		enum_GravaNomes.eAbreConexao: //abre conexao
			IF fbSQLDatabase2.Connect(INT_TO_UDINT(iNumeroDataBase)) THEN
				IF fbSQLDatabase2.bError THEN
					{error <'Não conseguiu abrir a conexao no banco do bloco FB_IniciaOsBlocosDeConfigDoMotor 1'>}
					IF fbSQLDatabase2.ipTcResult.ipSourceInfo.sName = 'ADSERR_DEVICE_LICENSENOTFOUND' THEN
						// se der isso ele nao fica tentando e gerando uma caralhada de erro pq nao tem a lisença
						eEstadoGrava := enum_GravaNomes.eParado;
					ELSE
						eEstadoGrava := enum_GravaNomes.eAbreConexao;
					END_IF
					
				ELSE
					IF fbSQLDatabase2.bConnected THEN
						eEstadoGrava := enum_GravaNomes.eCriaComando;
						xAberto := TRUE;
					ELSE
						eEstadoGrava := enum_GravaNomes.eFechaConexao;
						xAberto := FALSE;
					END_IF
				END_IF
			END_IF
			
		enum_GravaNomes.eCriaComando:
			IF fbSQLDatabase2.CreateCmd(ADR(fbSqlCommand)) THEN
				IF fbSQLDatabase2.bError THEN
					eEstadoGrava := enum_GravaNomes.eCriaComando;
				ELSE
					eEstadoGrava := enum_GravaNomes.eGravaNomes;
				END_IF
			END_IF
			
		enum_GravaNomes.eGravaNomes:
	
			//UPDATE `geral`.`iluminacaoconfig` SET `Tag` = 'IL' WHERE (`Telerruptor` = '1');
			
			Nome := stPM2100[iIndexGrava].config.sNomeFuncao;
			Tag := CONCAT(CONCAT('P', TO_STRING(iIndexGrava)), ' - ');
		
			IF FindAndReplace(
						pSrcString:= ADR(Nome), 
						pDeleteString:= ADR(Tag), 
						pInsertString:= ADR(Vazio), 
						pDstString:= ADR(Funcao), 
						nDstSize:= SIZEOF(Funcao)) = 0  THEN
						
				Funcao := '';	
			END_IF
						
			arrStr[1] := 'UPDATE dbexcelsior.';
			arrStr[2] := sNomeDataBase;
			arrStr[3] := ' SET Funcao = "';
			arrStr[4] := Funcao;
			arrStr[5] :='" WHERE (Medidor = "';
			arrStr[6] := TO_STRING(iIndexGrava);
			arrStr[7] := '");';
			
			sCmd2 := F_ConcatArray(sArray:= arrStr); 
	
			IF fbSQLCommand.Execute(pSQLCmd := ADR(sCmd2), cbSQLCmd := SIZEOF(sCmd2))
			THEN
				IF fbSQLCommand.bError THEN
					IF fbSQLCommand.ipTcResult.nEventId = 61 THEN
					// Esse erro acontece quando o database não tá criado, nesse caso ele tenta criar
						eEstadoGrava := enum_GravaNomes.eEsperando;
						xCriaTabela := TRUE;
					ELSE
						eEstadoGrava := enum_GravaNomes.eAbreConexao;
					END_IF
					sMensagemErro2 := 'Nao conseguiu a tag';
				ELSE
					sMensagemErro2	:= 'Conseguiu a tag';
				END_IF
				eEstadoGrava := enum_GravaNomes.eFechaConexao;
				iIndexGrava := 0;
			END_IF
			
		enum_GravaNomes.eFechaConexao:
			IF fbSQLDatabase2.Disconnect() THEN
		
				xGrava := FALSE;
				xLe := TRUE;
		
				eEstado := enum_LeituradosNomes.eEsperando;
				
				IF fbSQLDatabase2.bError THEN
					eEstadoGrava := enum_GravaNomes.eEsperando;
				ELSE
					eEstadoGrava := enum_GravaNomes.eEsperando;
					xAberto := FALSE;
				END_IF
			END_IF

END_CASE
END_ACTION

ACTION LeNomes:

CASE eEstado OF
		enum_LeituradosNomes.eEsperando: //Esperando
			IF xLe THEN
				eEstado := enum_LeituradosNomes.eAbreConexao;
			END_IF
			
		
		enum_LeituradosNomes.eAbreConexao: //abre conexao
			IF fbSqlDatabase.Connect(int_to_udint(iNumeroDataBase)) THEN
				IF fbSqlDatabase.bError THEN
					{error <'Não conseguiu abrir a conexao no banco do bloco FB_IniciaOsBlocosDeConfigDoMotor 1'>}
					IF fbSqlDatabase.ipTcResult.ipSourceInfo.sName = 'ADSERR_DEVICE_LICENSENOTFOUND' THEN
						// se der isso ele nao fica tentando e gerando uma caralhada de erro pq nao tem a lisença
						eEstado := enum_LeituradosNomes.eParado;
					ELSE
						eEstado := enum_LeituradosNomes.eAbreConexao;
					END_IF
					
				ELSE
					IF fbSqlDatabase.bConnected THEN
						eEstado := enum_LeituradosNomes.eLeOsNomes;
					END_IF
				END_IF
			END_IF
			
			enum_LeituradosNomes.eLeOsNomes: // le o role
				TagAProcurar		:= sTag1;
				stPara.eParaType	:= E_ExpParameterType.STRING_;
				stPara.nParaSize	:= SIZEOF(TagAProcurar);
				stPara.sParaName	:= 'Tag';
		
				diBaixo	:= LOWER_BOUND(stPM2100, 1);
				diCima		:= UPPER_BOUND(stPM2100, 1);
		
				// set command with placeholder
				sCmd := CONCAT(CONCAT('SELECT * FROM dbexcelsior.', sNomeDataBase), ';');
		
				// call functionblock
				IF fbPLCDBCmd.ExecuteDataReturn
					(
						hDBID := INT_TO_UDINT(iNumeroDataBase),
							pExpression := ADR(sCmd),
							cbExpression := SIZEOF(sCmd),
							pData := ADR(TagAProcurar),
							cbData := SIZEOF(TagAProcurar),
							pParameter := ADR(stPara),
							cbParameter := SIZEOF(stPara),
							nStartIndex := DINT_TO_UDINT(diBaixo),
							nRecordCount := DINT_TO_UDINT(diCima),
							pReturnData := ADR(EstruturaBancoLe),
							cbReturnData := SIZEOF(EstruturaBancoLe),
							pRecords := ADR(nRecords))
				THEN
					IF fbPLCDBCmd.bError THEN
						sMensagemErro1 := 'Nao conseguiu a tag';
						{error <'Não conseguiu ler o banco no bloco FB_IniciaOsBlocosDeConfigDoTelerruptor'>}
					ELSE
						sMensagemErro1	:= 'Conseguiu a tag';
						eEstado			:= enum_LeituradosNomes.eFechaConexao;
		
						FOR j := TO_INT(diBaixo) TO TO_INT(diCima) DO
							Anterior[j+1].config.sNomeFuncao := CONCAT(CONCAT(EstruturaBancoLe[j].Tag, ' - '), EstruturaBancoLe[j].Funcao);
							stPM2100[j+1].config.sNomeFuncao := CONCAT(CONCAT(EstruturaBancoLe[j].Tag, ' - '), EstruturaBancoLe[j].Funcao);
						END_FOR
						
					END_IF
				END_IF
			
			enum_LeituradosNomes.eFechaConexao: // FechaConexao conexao
				IF fbSqlDatabase.Disconnect() THEN
		
					xLe := FALSE;
					xInicia := FALSE;
		
					IF fbSqlDatabase.bError THEN
						{error <'Não conseguiu abrir a conexao no banco do bloco FB_IniciaOsBlocosDeConfigDoMotor 3'>}
						eEstado := enum_LeituradosNomes.eFechaConexao;
					ELSE
						eEstado := enum_LeituradosNomes.eMonitoraTrocaDeNomes;
					END_IF
				END_IF	

			enum_LeituradosNomes.eMonitoraTrocaDeNomes:
				FOR j := TO_INT(diBaixo) TO TO_INT(diCima) DO
					IF (stPM2100[j].config.sNomeFuncao <> Anterior[j].config.sNomeFuncao) THEN
						Anterior[j].config.sNomeFuncao := stPM2100[j].config.sNomeFuncao;
						iIndexGrava := j;
						xGrava := TRUE;
					END_IF
				END_FOR						
END_CASE
END_ACTION

END_FUNCTION_BLOCK

// FBs/MedicaoEnergia/FB_NomesMedidoresSEPAM
FUNCTION_BLOCK FB_NomesMedidoresSEPAM
VAR_IN_OUT
	stSEPAM	: ARRAY[*] OF st_SEPAMS20_Schneider;
END_VAR
VAR_INPUT
	xInicia			: BOOL;
	xCriaTabela		: BOOL;
	iNumeroDataBase	: INT		:= 1;
	sNomeDataBase	: STRING	:= 'nomes';
END_VAR
VAR_OUTPUT
	xOcupado	: BOOL;
END_VAR
VAR
	//Cria table
	rtCria			: R_TRIG;
	xCria			: BOOL;
	fbPLCDBCreate	: FB_PLCDBCreateEvt(sNetID := '', tTimeout := T#30S);
	ColumnInfo : ARRAY[0..2] OF ST_ColumnInfo := [(sName := 'Medidor', eType := E_ColumnType.Integer, nLength := 8, sProperty := 'IDENTITY(1,1)'),
												  (sName := 'Tag', eType := E_ColumnType.NVarChar, nLength := 80, sProperty := 'DEFAULT $'SEMTAG$''),
												  (sName := 'Funcao', eType := E_ColumnType.NVarChar, nLength := 80, sProperty := 'DEFAULT $'NADA$'')];
												  

	//Le os nomes
	xFirstScan		: BOOL := TRUE;
	xLe				: BOOL;
	sCmd			: STRING(1000);
	sTag1			: STRING;
	TagAProcurar	: STRING(80);
	sMensagemErro1	: STRING;
	iIndexGrava		: INT := 0;
	iAux			: DINT;
	diCima			: DINT;
	diBaixo			: DINT;
	nRecords		: UDINT;
	Anterior		: ARRAY[0..999] OF st_PM2100_485_Schneider;
	stPara			: ST_ExpParameter;
	EstruturaBancoLe: ARRAY[0..999] OF stConfigNomeMedidorDB;
	eEstado			: enum_LeituradosNomes := enum_LeituradosNomes.eEsperando;
	fbSQLDatabase	: FB_SQLDatabaseEvt(sNetID := '', tTimeout := T#30S);
	fbPLCDBCmd		: FB_PLCDBCmdEvt(sNetID := '', tTimeout := T#30S);
	
	
	//Gera os Telerruptores
	diParteBaixa		: DINT;
	diParteAlta			: DINT;
	i					: INT;
	xGeraMedidores		: BOOL;
	xEscreve			: BOOL;
	xEscreveAux			: BOOL;
	rtEscrita			: R_TRIG;	
	EstruturaBanco		: ARRAY[0..999] OF stConfigNomeMedidorDB;
	fbPLCDBWrite		: FB_PLCDBWriteEvt(sNetID := '', tTimeout := T#30S); //Bloco para gravar no banco de dados
	ColumnNamesGrava	: ARRAY[0..2] OF STRING(50) := ['Medidor',
														'Tag',
														'Funcao'
														];
	//Grava Nomes Novos
	j				: INT;
	xGrava			: BOOL;
	xAberto			: BOOL;
	sCmd2			: STRING(1000);
	sMensagemErro2	: STRING;
	Nome			: STRING;
	Vazio			: STRING := '';
	Tag				: STRING;
	Funcao			: STRING;
	arrStr			: ARRAY[1..10] OF STRING(255);
	eEstadoGrava	: enum_GravaNomes := enum_GravaNomes.eEsperando;
	fbSqlCommand		: FB_SQLCommandEvt(sNetID := '', tTimeout := T#30S);
	fbSQLDatabase2	: FB_SQLDatabaseEvt(sNetID := '', tTimeout := T#30S);
	
END_VAR



IF xFirstScan THEN
	xLe := TRUE;
	xCriaTabela := TRUE;
END_IF

IF xInicia THEN
	xLe := TRUE;
	eEstado := enum_LeituradosNomes.eEsperando;
END_IF




GeraTabela();
//GeraOsMedidores();
LeNomes();
GravaValores();

xFirstScan := FALSE;

ACTION GeraOsMedidores:

diParteBaixa	:= LOWER_BOUND(stSEPAM, 1);
diParteAlta		:= UPPER_BOUND(stSEPAM, 1);

IF xGeraMedidores THEN

	xEscreve := TRUE;
	rtEscrita(CLK := xEscreve, Q =>);

	IF rtEscrita.q THEN
		xEscreveAux						:= TRUE;
		xOcupado						:= TRUE;
		i := DINT_TO_INT(diParteBaixa);
	END_IF

	IF xEscreveAux THEN
		EstruturaBanco[i].Tag := CONCAT('P', INT_TO_STRING(i+1));
		EstruturaBanco[i].Medidor := INT_TO_DINT(i);
		
		IF fbPLCDBWrite.WriteStruct
		(
			hDBID := INT_TO_UDINT(iNumeroDataBase),
				sTableName := sNomeDataBase,
				pRecord := ADR(EstruturaBanco[i]),
				cbRecord := SIZEOF(EstruturaBanco[i]),
				pColumnNames := ADR(ColumnNamesGrava),
				cbColumnNames := SIZEOF(ColumnNamesGrava))
		THEN
			i := i +1;
		ELSE
			IF fbPLCDBWrite.bError THEN
				IF fbPLCDBWrite.ipTcResult.nEventId = 61 THEN
					xCriaTabela := TRUE;
				END_IF
			END_IF
		END_IF
		
		IF i > diParteAlta THEN
			xOcupado	:= FALSE;
			xEscreve 	:= FALSE;
			rtEscrita(CLK := xEscreve, Q =>);
			xEscreveAux	:= FALSE;
			xGeraMedidores := FALSE;
			i := DINT_TO_INT(diParteBaixa);
			
			xLe := TRUE;
			eEstado := enum_LeituradosNomes.eEsperando;
		END_IF

	END_IF
END_IF
END_ACTION

ACTION GeraTabela:

rtCria(CLK := xCriaTabela, Q =>);

IF rtCria.q THEN
	xCria		:= TRUE;
	xOcupado	:= TRUE;
END_IF

IF xCria THEN

	IF fbPLCDBCreate.Table
		(
			hDBID := INT_TO_UDINT(iNumeroDataBase),
				sTableName := sNomeDataBase,
				pTableCfg := ADR(ColumnInfo),
				cbTableCfg := SIZEOF(ColumnInfo))
	THEN
		xCria		:= FALSE;
		xCriaTabela	:= FALSE;
		xOcupado	:= FALSE;
		xGeraMedidores	:= TRUE;
		i			:= 0;
	END_IF

END_IF
END_ACTION

ACTION GravaValores:
CASE eEstadoGrava OF
		enum_GravaNomes.eEsperando: //Esperando
			IF xGrava THEN
				IF xAberto THEN
					eEstadoGrava := enum_GravaNomes.eCriaComando;
				ELSE
					eEstadoGrava := enum_GravaNomes.eAbreConexao;
				END_IF
				
			END_IF
			
		enum_GravaNomes.eAbreConexao: //abre conexao
			IF fbSQLDatabase2.Connect(INT_TO_UDINT(iNumeroDataBase)) THEN
				IF fbSQLDatabase2.bError THEN
					{error <'Não conseguiu abrir a conexao no banco do bloco FB_IniciaOsBlocosDeConfigDoMotor 1'>}
					IF fbSQLDatabase2.ipTcResult.ipSourceInfo.sName = 'ADSERR_DEVICE_LICENSENOTFOUND' THEN
						// se der isso ele nao fica tentando e gerando uma caralhada de erro pq nao tem a lisença
						eEstadoGrava := enum_GravaNomes.eParado;
					ELSE
						eEstadoGrava := enum_GravaNomes.eAbreConexao;
					END_IF
					
				ELSE
					IF fbSQLDatabase2.bConnected THEN
						eEstadoGrava := enum_GravaNomes.eCriaComando;
						xAberto := TRUE;
					ELSE
						eEstadoGrava := enum_GravaNomes.eFechaConexao;
						xAberto := FALSE;
					END_IF
				END_IF
			END_IF
			
		enum_GravaNomes.eCriaComando:
			IF fbSQLDatabase2.CreateCmd(ADR(fbSqlCommand)) THEN
				IF fbSQLDatabase2.bError THEN
					eEstadoGrava := enum_GravaNomes.eCriaComando;
				ELSE
					eEstadoGrava := enum_GravaNomes.eGravaNomes;
				END_IF
			END_IF
			
		enum_GravaNomes.eGravaNomes:
	
			//UPDATE `geral`.`iluminacaoconfig` SET `Tag` = 'IL' WHERE (`Telerruptor` = '1');
			
			Nome := stSEPAM[iIndexGrava].config.sNomeFuncao;
			Tag := CONCAT(CONCAT('P', TO_STRING(iIndexGrava)), ' - ');
		
			IF FindAndReplace(
						pSrcString:= ADR(Nome), 
						pDeleteString:= ADR(Tag), 
						pInsertString:= ADR(Vazio), 
						pDstString:= ADR(Funcao), 
						nDstSize:= SIZEOF(Funcao)) = 0  THEN
						
				Funcao := '';	
			END_IF
						
			arrStr[1] := 'UPDATE dbexcelsior.';
			arrStr[2] := sNomeDataBase;
			arrStr[3] := ' SET Funcao = "';
			arrStr[4] := Funcao;
			arrStr[5] :='" WHERE (Medidor = "';
			arrStr[6] := TO_STRING(iIndexGrava);
			arrStr[7] := '");';
			
			sCmd2 := F_ConcatArray(sArray:= arrStr); 
	
			IF fbSQLCommand.Execute(pSQLCmd := ADR(sCmd2), cbSQLCmd := SIZEOF(sCmd2))
			THEN
				IF fbSQLCommand.bError THEN
					IF fbSQLCommand.ipTcResult.nEventId = 61 THEN
					// Esse erro acontece quando o database não tá criado, nesse caso ele tenta criar
						eEstadoGrava := enum_GravaNomes.eEsperando;
						xCriaTabela := TRUE;
					ELSE
						eEstadoGrava := enum_GravaNomes.eAbreConexao;
					END_IF
					sMensagemErro2 := 'Nao conseguiu a tag';
				ELSE
					sMensagemErro2	:= 'Conseguiu a tag';
				END_IF
				eEstadoGrava := enum_GravaNomes.eFechaConexao;
				iIndexGrava := 0;
			END_IF
			
		enum_GravaNomes.eFechaConexao:
			IF fbSQLDatabase2.Disconnect() THEN
		
				xGrava := FALSE;
				xLe := TRUE;
		
				eEstado := enum_LeituradosNomes.eEsperando;
				
				IF fbSQLDatabase2.bError THEN
					eEstadoGrava := enum_GravaNomes.eEsperando;
				ELSE
					eEstadoGrava := enum_GravaNomes.eEsperando;
					xAberto := FALSE;
				END_IF
			END_IF

END_CASE
END_ACTION

ACTION LeNomes:

CASE eEstado OF
		enum_LeituradosNomes.eEsperando: //Esperando
			IF xLe THEN
				eEstado := enum_LeituradosNomes.eAbreConexao;
			END_IF
			
		
		enum_LeituradosNomes.eAbreConexao: //abre conexao
			IF fbSqlDatabase.Connect(int_to_udint(iNumeroDataBase)) THEN
				IF fbSqlDatabase.bError THEN
					{error <'Não conseguiu abrir a conexao no banco do bloco FB_IniciaOsBlocosDeConfigDoMotor 1'>}
					IF fbSqlDatabase.ipTcResult.ipSourceInfo.sName = 'ADSERR_DEVICE_LICENSENOTFOUND' THEN
						// se der isso ele nao fica tentando e gerando uma caralhada de erro pq nao tem a lisença
						eEstado := enum_LeituradosNomes.eParado;
					ELSE
						eEstado := enum_LeituradosNomes.eAbreConexao;
					END_IF
					
				ELSE
					IF fbSqlDatabase.bConnected THEN
						eEstado := enum_LeituradosNomes.eLeOsNomes;
					END_IF
				END_IF
			END_IF
			
			enum_LeituradosNomes.eLeOsNomes: // le o role
				TagAProcurar		:= sTag1;
				stPara.eParaType	:= E_ExpParameterType.STRING_;
				stPara.nParaSize	:= SIZEOF(TagAProcurar);
				stPara.sParaName	:= 'Tag';
		
				diBaixo	:= LOWER_BOUND(stSEPAM, 1);
				diCima		:= UPPER_BOUND(stSEPAM, 1);
		
				// set command with placeholder
				sCmd := CONCAT(CONCAT('SELECT * FROM dbexcelsior.', sNomeDataBase), ';');
		
				// call functionblock
				IF fbPLCDBCmd.ExecuteDataReturn
					(
						hDBID := INT_TO_UDINT(iNumeroDataBase),
							pExpression := ADR(sCmd),
							cbExpression := SIZEOF(sCmd),
							pData := ADR(TagAProcurar),
							cbData := SIZEOF(TagAProcurar),
							pParameter := ADR(stPara),
							cbParameter := SIZEOF(stPara),
							nStartIndex := DINT_TO_UDINT(diBaixo-1),
							nRecordCount := DINT_TO_UDINT(diCima),
							pReturnData := ADR(EstruturaBancoLe),
							cbReturnData := SIZEOF(EstruturaBancoLe),
							pRecords := ADR(nRecords))
				THEN
					IF fbPLCDBCmd.bError THEN
						sMensagemErro1 := 'Nao conseguiu a tag';
						{error <'Não conseguiu ler o banco no bloco FB_IniciaOsBlocosDeConfigDoTelerruptor'>}
					ELSE
						sMensagemErro1	:= 'Conseguiu a tag';
						eEstado			:= enum_LeituradosNomes.eFechaConexao;
		
						FOR j := TO_INT(diBaixo) TO TO_INT(diCima) DO
							Anterior[j].config.sNomeFuncao := CONCAT(CONCAT(EstruturaBancoLe[j-129].Tag, ' - '), EstruturaBancoLe[j-129].Funcao);
							stSEPAM[j].config.sNomeFuncao := CONCAT(CONCAT(EstruturaBancoLe[j-129].Tag, ' - '), EstruturaBancoLe[j-129].Funcao);
						END_FOR
						
					END_IF
				END_IF
			
			enum_LeituradosNomes.eFechaConexao: // FechaConexao conexao
				IF fbSqlDatabase.Disconnect() THEN
		
					xLe := FALSE;
					xInicia := FALSE;
		
					IF fbSqlDatabase.bError THEN
						{error <'Não conseguiu abrir a conexao no banco do bloco FB_IniciaOsBlocosDeConfigDoMotor 3'>}
						eEstado := enum_LeituradosNomes.eFechaConexao;
					ELSE
						eEstado := enum_LeituradosNomes.eMonitoraTrocaDeNomes;
					END_IF
				END_IF	

			enum_LeituradosNomes.eMonitoraTrocaDeNomes:
				FOR j := TO_INT(diBaixo) TO TO_INT(diCima) DO
					IF (stSEPAM[j].config.sNomeFuncao <> Anterior[j].config.sNomeFuncao) THEN
						Anterior[j].config.sNomeFuncao := stSEPAM[j].config.sNomeFuncao;
						iIndexGrava := j;
						xGrava := TRUE;
					END_IF
				END_FOR						
END_CASE
END_ACTION

END_FUNCTION_BLOCK

// FBs/MedicaoEnergia/FB_SalvaDadosMedidores
FUNCTION_BLOCK FB_SalvaDadosMedidores
VAR_INPUT
	xCriaTabelas		: BOOL;				// tenta criar a tabela
	iNumeroDataBase		: INT	:= 1;		// id do database
	iMedidor			: INT;
	xMedidorOnline		: BOOL;
	rCorrenteA			: REAL;
	rCorrenteB			: REAL;
	rCorrenteC			: REAL;
	rCorrenteMedia		: REAL;
	stHoraAgora			: TIMESTRUCT;
END_VAR
VAR_OUTPUT
	xOcupado 				: BOOL;
	iEndereco				: INT;
END_VAR
VAR
	//Cria table
	rtCria				: R_TRIG;
	xComecaCriarTabelas	: BOOL;
	fbPLCDBCreate1	: FB_PLCDBCreateEvt(sNetID := '', tTimeout := T#30S);
	
	ColumnInfo1 : ARRAY[0..5] OF ST_ColumnInfo := [	(sName := 'rCorrenteA',	eType := E_ColumnType.REAL_,	nLength := 4),
												(sName := 'rCorrenteB',	eType := E_ColumnType.REAL_,	nLength := 4),
												(sName := 'rCorrenteC',	eType := E_ColumnType.REAL_,	nLength := 4),
												(sName := 'rCorrenteMedia',	eType := E_ColumnType.REAL_,	nLength := 4),
												(sName := 'medidor',	eType := E_ColumnType.Integer, 	nLength := 2),
												(sName := 'timestamps', 	eType := E_ColumnType.DateTime, nLength := 4, sProperty := 'DEFAULT CURRENT_TIMESTAMP ON UPDATE CURRENT_TIMESTAMP')];
												
	//Grava valores
	xEscreve			: BOOL;
	rtEscreve			: R_TRIG;
	tonEscrita			: TON;
	arString			: ARRAY[0..6] OF STRING(255);
	fbSqlCommand		: FB_SQLCommandEvt(sNetID := '', tTimeout := T#30S);
	fbSQLDatabase		: FB_SQLDatabaseEvt(sNetID := '', tTimeout := T#30S);
	sCmd				: STRING(1000);
	sMensagemErro1 		: STRING;
	xAberto 			: BOOL;
	rtComecaEscrever 	: R_TRIG;
	iEstado 			: INT := 1;
	i					: INT;
	
END_VAR

//Criado Por Augusto Cazzanelli para o Projeto Excelsior
IF xLicensaValida651641iih THEN
	GeraTabela();
	
	iEndereco := iMedidor;
	
	rtEscreve(CLK:= stHoraAgora.wMinute MOD 5 = 0, Q=> );
	
	IF rtEscreve.Q THEN
		xEscreve := TRUE;
	END_IF
	
	GravaValores();
END_IF

ACTION GeraTabela:

rtCria(CLK := xCriaTabelas, Q =>);

IF rtCria.q THEN
	xComecaCriarTabelas		:= TRUE;
	xOcupado				:= TRUE;
END_IF

IF xComecaCriarTabelas THEN
		//Cria a tabela com os minutos inidividuais de cada um dos 15 min
		IF fbPLCDBCreate1.Table
			(
				hDBID := INT_TO_UDINT(iNumeroDataBase),
					sTableName := 'corrente',
					pTableCfg := ADR(ColumnInfo1),
					cbTableCfg := SIZEOF(ColumnInfo1))
		THEN
			xComecaCriarTabelas		:= FALSE;
			xCriaTabelas	:= FALSE;
			xOcupado := FALSE;
		END_IF
ELSE
	xOcupado := FALSE;
END_IF
END_ACTION

ACTION GravaValores:

CASE iEstado OF
	1: //Esperando
		IF xEscreve AND xMedidorOnline THEN
			IF xAberto THEN
				iEstado := 3;	//Caso para abrir a conexão
			ELSE
				iEstado := 2;	//Caso em que a conexão já foi aberta
			END_IF
		END_IF
		
	2: //abre conexao
		IF fbSqlDatabase.Connect(int_to_udint(iNumeroDataBase)) THEN
			IF fbSqlDatabase.bError THEN
				IF fbSqlDatabase.ipTcResult.nEventId = 1828 THEN
					// se der isso ele nao fica tentando e gerando uma caralhada de erro pq nao tem a lisença
					iEstado := 0;
				ELSE
					iEstado := 2;
				END_IF
			ELSE
				IF fbSqlDatabase.bConnected THEN
					iEstado := 3;
					xAberto := TRUE;
				ELSE
					iEstado := 5;
					xAberto := FALSE;
				END_IF
			END_IF
		END_IF
		
	3:
		IF fbSqlDatabase.CreateCmd(ADR(fbSqlCommand)) THEN
			IF fbSqlDatabase.bError THEN
				iEstado := 3;
			ELSE
				iEstado := 4;
			END_IF
		END_IF
		
		4: // le o role
		//'INSERT INTO dbexcelsior.minutos(rDemanda1min,medidor) VALUES (rDemanda1min, iMedidor);'	
		
		FOR i := 0 TO 3 DO
			arString[i] := '';
		END_FOR
	
		IF xMedidorOnline THEN
			arString[0] := 'INSERT INTO dbexcelsior.corrente(rCorrenteA,rCorrenteB,rCorrenteC,rCorrenteMedia,medidor) VALUES (';
			arString[1] := CONCAT(TO_STRING(rCorrenteA),',');
			arString[2] := CONCAT(TO_STRING(rCorrenteB),',');
			arString[3] := CONCAT(TO_STRING(rCorrenteC),',');
			arString[4] := CONCAT(TO_STRING(rCorrenteMedia),',');
			arString[5] := CONCAT(TO_STRING(iMedidor),');');
		END_IF

	
		sCmd := F_ConcatArray(sArray:= arString);
		
		IF fbSQLCommand.Execute(pSQLCmd := ADR(sCmd), cbSQLCmd := SIZEOF(sCmd)) THEN
			IF fbSQLCommand.bError THEN
				IF fbSQLCommand.ipTcResult.nEventId = 61 THEN
				// Esse erro acontece quando o database não tá criado, nesse caso ele tenta criar
				iEstado := 1;
					xCriaTabelas := TRUE;
				ELSE
					iEstado := 2;
				END_IF
				sMensagemErro1 := 'Nao conseguiu a tag';
			ELSE
				sMensagemErro1	:= 'Conseguiu a tag';
			END_IF
			iEstado := 5;
			xEscreve			:= FALSE;
		END_IF
		
		
	5: // FechaConexao conexao
			IF fbSqlDatabase.Disconnect() THEN
	
				xEscreve			:= FALSE;
	
				IF fbSqlDatabase.bError THEN
					iEstado := 1;
				ELSE
					iEstado := 1;
					xAberto := FALSE;
				END_IF
			END_IF
END_CASE
END_ACTION

END_FUNCTION_BLOCK

// FBs/Partidas/KPI/FB_KPIPartidasSQL
FUNCTION_BLOCK FB_KPIPartidasSQL
VAR_IN_OUT
	Motores : ARRAY[*] OF st_Partida;
END_VAR
VAR_INPUT
	tTempoDeAmostra : TIME;
	xCriaTabela : BOOL;
	iNumeroDataBase : INT := 1;
	sNomeTabela : STRING := 'KPIMotores';
	stHoraAgora : TIMESTRUCT;
	xFazAgora : BOOL;
END_VAR
VAR_OUTPUT
	xGravando : BOOL;
	iRegistro : INT;
END_VAR
VAR
	iEstado : INT := 1;
	rtCria : R_TRIG;
	xCria : BOOL;
	fbPLCDBCreate : FB_PLCDBCreateEvt(sNetID:='', tTimeout:=T#30S);
	
	ColumnInfo : ARRAY[0..7] OF ST_ColumnInfo := [(sName := 'ID', eType := E_ColumnType.BigInt, nLength := 8, sProperty := 'IDENTITY(1,1)'),
												(sName := 'TAG', eType := E_ColumnType.NVarChar, nLength := 80),
												(sName := 'Desligado', eType := E_ColumnType.REAL_, nLength := 8),
												(sName := 'Ligado', eType := E_ColumnType.REAL_, nLength := 8),
												(sName := 'Emergencia', eType := E_ColumnType.REAL_, nLength := 8),
												(sName := 'Falha', eType := E_ColumnType.REAL_, nLength := 8),
												(sName := 'Interlock', eType := E_ColumnType.REAL_, nLength := 8),
												(
				sName := 'Timestamp',
					eType := E_ColumnType.DateTime,
					nLength := 4,
					sProperty :='DEFAULT CURRENT_TIMESTAMP ON UPDATE CURRENT_TIMESTAMP')];
	
	tonEscrita : TON;
	xEscreve : BOOL;
	
	xAtualiza : BOOL;
	ColumnNames : ARRAY[0..6] OF STRING(50) := ['ID',
												'TAG',
												'Desligado',
												'Ligado',
												'Emergencia',
												'Falha',
												'Interlock'];
	iTamanhoHistorico : DINT;
	
	i : INT;
	
	fbPLCDBWrite : FB_PLCDBWriteEvt(sNetID:='', tTimeout:=T#30S); //Bloco para gravar no banco de dados
	sMensagemErroEscrita : STRING;
	
	AuxEscreve : ARRAY[1..500] OF st_KPISQL;
	
	wHoraAnterior : WORD;
	xFirstScan : BOOL := TRUE;
	iMax : INT;
	iMin : INT;
END_VAR



IF xFirstScan THEN
	iMax := DINT_TO_INT(UPPER_BOUND(Motores,1));
	iMin := DINT_TO_INT(LOWER_BOUND(Motores,1));
	
	wHoraAnterior 	:= stHoraAgora.wHour;
END_IF


IF (stHoraAgora.wHour <> wHoraAnterior AND stHoraAgora.wMinute = 2) OR xFazAgora AND NOT xGravando THEN
	
	FOR i := iMin + 1 TO iMax DO
		IF Motores[i].KPI[1].rPorcDesligado > 0.01 THEN
			AuxEscreve[i].Desligado := Motores[i].KPI[1].rPorcDesligado;
		ELSE
			AuxEscreve[i].Desligado := 0;
		END_IF
		
		IF Motores[i].KPI[1].rPorcEmergencia > 0.01 THEN
			AuxEscreve[i].Emergencia := Motores[i].KPI[1].rPorcEmergencia;
		ELSE
			AuxEscreve[i].Emergencia := 0;
		END_IF
		
		IF Motores[i].KPI[1].rPorcFalha > 0.01 THEN
			AuxEscreve[i].Falha := Motores[i].KPI[1].rPorcFalha;
		ELSE
			AuxEscreve[i].Falha := 0;
		END_IF
		
		IF Motores[i].KPI[1].rPorcInterlock > 0.01 THEN
			AuxEscreve[i].Interlock := Motores[i].KPI[1].rPorcInterlock;
		ELSE
			AuxEscreve[i].Interlock := 0;
		END_IF
		
		IF Motores[i].KPI[1].rPorcLigado > 0.01 THEN
			AuxEscreve[i].Ligado := Motores[i].KPI[1].rPorcLigado;
		ELSE
			AuxEscreve[i].Ligado := 0;
		END_IF
		
		IF Motores[iMax].BancoDeDados.Tag <> '' THEN
			AuxEscreve[i].TAG := Motores[i].BancoDeDados.Tag;
		ELSE
			//se nao tiver tag pula fora pra nao ficar rodando onde nao precisa
			EXIT;
		END_IF
	END_FOR

	wHoraAnterior 	:= stHoraAgora.wHour;
	xEscreve		:= TRUE;
	xFazAgora		:= FALSE;
	xGravando 		:= TRUE;
	iRegistro		:= iMin + 1;
END_IF

IF xGravando AND NOT xEscreve THEN
	iRegistro := iRegistro + 1;
	xEscreve := TRUE;
	IF AuxEscreve[iRegistro].TAG = '' THEN
		xGravando := FALSE;
		xEscreve := FALSE;
	END_IF
END_IF

GeraTabela();
GravaHistorico();


xFirstScan := false;

ACTION GeraTabela:

rtCria(CLK := xCriaTabela, Q =>);

IF rtCria.q THEN
	xCria := TRUE;
END_IF

IF xCria THEN

	IF fbPLCDBCreate.Table(
			hDBID := INT_TO_UDINT(iNumeroDataBase),
			sTableName := sNomeTabela,
			pTableCfg := ADR(ColumnInfo),
			cbTableCfg := SIZEOF(ColumnInfo))
	THEN
		xCria := FALSE;
		xCriaTabela := FALSE;
	END_IF

END_IF
END_ACTION

ACTION GravaHistorico:




IF xEscreve THEN
	IF fbPLCDBWrite.WriteStruct(
			hDBID := int_to_Udint(iNumeroDataBase),
			sTableName := sNomeTabela,
			pRecord := ADR(AuxEscreve[iRegistro]),
			cbRecord := SIZEOF(AuxEscreve[iRegistro]),
			pColumnNames := ADR(ColumnNames),
			cbColumnNames := SIZEOF(ColumnNames))
	THEN
		IF fbPLCDBWrite.bError THEN
			sMensagemErroEscrita := 'Erro ao gravar no banco de dados';
			xEscreve             := FALSE;
		ELSE
			sMensagemErroEscrita := 'Dados gravados com sucesso';
			xEscreve             := FALSE;
		END_IF
	END_IF
END_IF
END_ACTION

END_FUNCTION_BLOCK

// FBs/Partidas/SalvaUsoNormal/FB_BDMotores
//{attribute 'hide_all_locals'}
FUNCTION_BLOCK FB_BDMotores
VAR_IN_OUT
	iAtualizandoAtual : INT;
END_VAR
VAR_INPUT
	Motor		: st_Partida;	// st do motor pra pegar os dados
	Nome		: STRING;		// nome do motor para a criação da tabela
	xCriaTabela	: BOOL;			// tenta criar a tabela
	HoraAgora	: TIMESTRUCT;	// pra saber quando gravar
	sCaminhoCSV	: STRING;		// caminho pro CSV
	iMaxAtualizando			: INT := 50;
END_VAR
VAR_OUTPUT
END_VAR
VAR
	// cria tabela
	xCria			: BOOL;
	rtCria			: R_TRIG;
	fbPLCDBCreate	: FB_PLCDBCreateEvt(sNetID := '', tTimeout := T#5S);

	ColumnInfo : ARRAY[0..9] OF ST_ColumnInfo := [(sName := 'ID', eType := E_ColumnType.BigInt, nLength := 8, sProperty := 'IDENTITY(1,1)'),
												(sName := 'Velocidade', eType := E_ColumnType.SmallInt, nLength := 2),
												(sName := 'Corrente', eType := E_ColumnType.REAL_, nLength := 4),
												(sName := 'TemperaturaDoMotor', eType := E_ColumnType.REAL_, nLength := 4),
												(sName := 'Torque', eType := E_ColumnType.REAL_, nLength := 4),
												(sName := 'StatusIHM', eType := E_ColumnType.NVarChar, nLength := 80),
												(sName := 'HorimetroD', eType := E_ColumnType.NVarChar, nLength := 80),
												(sName := 'TotalDePartidas', eType := E_ColumnType.SmallInt, nLength := 2),
												(sName := 'TotalDeFalhas', eType := E_ColumnType.SmallInt, nLength := 2),
												(
				sName := 'Timestamp',
					eType := E_ColumnType.DateTime,
					nLength := 4,
					sProperty := 'DEFAULT CURRENT_TIMESTAMP ON UPDATE CURRENT_TIMESTAMP')];

	// escreve na tabela
	fbPLCDBWrite	: FB_PLCDBWriteEvt(sNetID := '', tTimeout := T#5S);
	ValorPraEscrita	: st_EscritaBD;

	ColumnNames : ARRAY[0..8] OF STRING(50) := ['ID',
												'Velocidade',
												'Corrente',
												'TemperaturaDoMotor',
												'Torque',
												'StatusIHM',
												'HorimetroD',
												'TotalDePartidas',
												'TotalDeFalhas'];

	tUltimoHorimeto	: TIME;
	xEscreve		: BOOL;

	// guarda para escrever o ultimo minuto CSV
	HistoricoDoMinuto : ARRAY[0..59] OF st_EscritaBD;

	rtMudouMinuto	: R_TRIG;
	rtMudouSegundo	: R_TRIG;

	UltimaHora : TIMESTRUCT;

	rtMudouFalhas	: R_TRIG;
	rtMudouPartidas	: R_TRIG;

	iUltimaFalha	: INT;
	iUltimaPartida	: INT;

	rtTrocouDia : R_TRIG;

	//Escrita do CSV
	rtEntrouEmFalha : R_TRIG;

	FBEscreveCSV		: FB_EscreveCSV;
	fbCriaEstruta		: FB_CreateDir;
	dataBase			: ARRAY[0..60, 0..7] OF STRING(255);
	sCaminhoPasta		: STRING;
	sNomeEcaminho		: STRING;
	rtTerminouDeCriar	: R_TRIG;

	sAux : ARRAY[0..25] OF STRING(255);

	i	: INT;
	j	: INT;
	
	xOlhaSeTemEspacoConexao : BOOL;
	rt_TemEspeco : R_TRIG;
	
END_VAR


GeraTabela();

AtualizaValor();

EscreveCSV();

rtMudouMinuto(CLK := tUltimoHorimeto + T#1M = Motor.Sa.tHorimetro, Q =>);

// ve se mudou pra jogar no banco
IF rtMudouMinuto.q AND Motor.Sa.xCmdFwd THEN
	xEscreve		:= TRUE;
	xOlhaSeTemEspacoConexao := FALSE;
	tUltimoHorimeto	:= Motor.Sa.tHorimetro;
END_IF

// se tem espaço pra atualizar ele vai la
rt_TemEspeco(CLK:= xEscreve AND iAtualizandoAtual < iMaxAtualizando, Q=> );
IF rt_TemEspeco.q THEN
	xOlhaSeTemEspacoConexao := TRUE;
	iAtualizandoAtual := iAtualizandoAtual + 1;
END_IF

IF xOlhaSeTemEspacoConexao THEN
	IF fbPLCDBWrite.WriteStruct
		(
			hDBID := 1,
				sTableName := nome,
				pRecord := ADR(ValorPraEscrita),
				cbRecord := SIZEOF(ValorPraEscrita),
				pColumnNames := ADR(ColumnNames),
				cbColumnNames := SIZEOF(ColumnNames))
	THEN
		xEscreve := FALSE;
		xOlhaSeTemEspacoConexao := FALSE;
		iAtualizandoAtual := iAtualizandoAtual - 1;
	END_IF
END_IF

rtMudouSegundo(CLK := HoraAgora.wSecond <> UltimaHora.wSecond, Q =>);

IF rtMudouSegundo.q THEN
	i := WORD_TO_INT(HoraAgora.wSecond);
	HistoricoDoMinuto[i] := ValorPraEscrita;
END_IF

UltimaHora := HoraAgora;

ACTION AtualizaValor:

ValorPraEscrita.Corrente			:= Motor.Sa.rCorrente;
ValorPraEscrita.Velocidade			:= Motor.Sa.iVelocidade;
ValorPraEscrita.TemperaturaDoMotor	:= Motor.Sa.rTemperaturaMotor;
ValorPraEscrita.Torque				:= Motor.Sa.rTorque;

ValorPraEscrita.HorimetroD := Motor.Sa.sHorimetro;

//se tiver em falha ele manda o erro pra BD, se nao manda o status atual dele
IF Motor.Sa.xFalha THEN
	ValorPraEscrita.StatusIHM := Motor.LeiturasInversorIHM.sUltimoErro;
ELSE
	ValorPraEscrita.StatusIHM := Motor.LeiturasInversorIHM.sStatusConexao;
END_IF

// se eles forem diferente e ele for maior que 1 incrementa o numero de falhas, é assim pq o cara pode dar reset no contador
rtMudouFalhas(CLK := ((iUltimaFalha <> Motor.Sa.iFalhaPartida) AND Motor.Sa.iFalhaPartida > 0), Q =>);

IF rtMudouFalhas.q THEN
	ValorPraEscrita.TotalDeFalhas := ValorPraEscrita.TotalDeFalhas + 1;
END_IF

iUltimaFalha := Motor.Sa.iFalhaPartida;

rtMudouPartidas(CLK := (iUltimaPartida <> Motor.Sa.iPartidas) AND Motor.Sa.iPartidas > 0, Q =>);

IF rtMudouPartidas.q THEN
	ValorPraEscrita.TotalDePartidas := ValorPraEscrita.TotalDePartidas + 1;
END_IF

iUltimaPartida := Motor.Sa.iPartidas;

rtTrocouDia(CLK := HoraAgora.wDay <> UltimaHora.wDay, Q =>);

IF rtTrocouDia.q THEN
	ValorPraEscrita.TotalDeFalhas	:= 0;
	ValorPraEscrita.TotalDePartidas	:= 0;
	tUltimoHorimeto					:= Motor.Sa.tHorimetro;
END_IF
END_ACTION

ACTION EscreveCSV:

rtEntrouEmFalha(CLK := Motor.Sa.xFalha AND ValorPraEscrita.StatusIHM <> 'Carregando', Q =>);

IF rtEntrouEmFalha.q THEN
	
	//Pra no segundo de agora pegar a falha
	i := WORD_TO_INT(HoraAgora.wSecond);
	HistoricoDoMinuto[i] := ValorPraEscrita;


	//Ajeita o data base
	dataBase[0, 0]	:= 'Velocidade';
	dataBase[0, 1]	:= 'Corrente';
	dataBase[0, 2]	:= 'TemperaturaDoMotor';
	dataBase[0, 3]	:= 'Torque';
	dataBase[0, 4]	:= 'StatusIHM';
	dataBase[0, 5]	:= 'HorimetroD';
	dataBase[0, 6]	:= 'TotalDePartidas';
	dataBase[0, 7]	:= 'TotalDeFalhas';

	FOR i := 1 TO 60 DO
		FOR J := 0 TO 8 DO
			CASE j OF
				0:
					dataBase[i, j] := TO_STRING(HistoricoDoMinuto[i - 1].Velocidade);

				1:
					dataBase[i, j] := TO_STRING(HistoricoDoMinuto[i - 1].Corrente);

				2:
					dataBase[i, j] := TO_STRING(HistoricoDoMinuto[i - 1].TemperaturaDoMotor);

				3:
					dataBase[i, j] := TO_STRING(HistoricoDoMinuto[i - 1].Torque);

				4:
					dataBase[i, j] := TO_STRING(HistoricoDoMinuto[i - 1].StatusIHM);

				5:
					dataBase[i, j] := TO_STRING(HistoricoDoMinuto[i - 1].HorimetroD);

				6:
					dataBase[i, j] := TO_STRING(HistoricoDoMinuto[i - 1].TotalDePartidas);

				7:
					dataBase[i, j] := TO_STRING(HistoricoDoMinuto[i - 1].TotalDeFalhas);
			END_CASE
		END_FOR
	END_FOR

	//Ve se a pasta ta criada certa 

	fbCriaEstruta(bExecute := TRUE);

	//Ajeita o nome
	sAux[1]			:= sCaminhoCSV;
	sAux[2]			:= '\Falha_';
	sAux[3]			:= Nome;
	sCaminhoPasta	:= CONCAT(sCaminhoCSV, CONCAT('\Falha_', Nome));

	sAux[1]		:= sCaminhoPasta;
	sAux[2]		:= '\';
	sAux[3]		:= TO_STRING(HoraAgora.wYear);
	sAux[4]		:= 'A_';
	sAux[5]		:= TO_STRING(HoraAgora.wMonth);
	sAux[6]		:= 'M_';
	sAux[7]		:= TO_STRING(HoraAgora.wDay);
	sAux[8]		:= 'D_';
	sAux[9]		:= TO_STRING(HoraAgora.wHour);
	sAux[10]	:= 'h_';
	sAux[11]	:= TO_STRING(HoraAgora.wMinute);
	sAux[12]	:= 'm_';
	sAux[13]	:= TO_STRING(HoraAgora.wSecond);
	sAux[20]	:= '.csv';

	sNomeEcaminho := F_ConcatArray(sAux);
END_IF

fbCriaEstruta
	(
		sPathName := sCaminhoPasta,
			ePath := PATH_GENERIC,
			tTimeout := T#5S,
			bBusy =>);

rtTerminouDeCriar(CLK := NOT fbCriaEstruta.bBusy, Q =>);

IF rtTerminouDeCriar.q THEN
	fbCriaEstruta(bExecute := FALSE);
	FBEscreveCSV.bInicia := TRUE;
END_IF

FBEscreveCSV
	(
		sCaminhoENome := sNomeEcaminho,
			xEscrevePorCima := FALSE,
			database := dataBase,
			bBusy =>,
			bError =>,
			nErrId =>,
			iTotal =>,
			iAgora =>);

IF NOT FBEscreveCSV.bBusy THEN
	FBEscreveCSV.bInicia := FALSE;
END_IF
END_ACTION

ACTION GeraTabela:

rtCria(CLK := xCriaTabela, Q =>);

IF rtCria.q THEN
	xCria := TRUE;
END_IF

IF xCria THEN

	IF fbPLCDBCreate.Table
		(
			hDBID := 1,
				sTableName := nome,
				pTableCfg := ADR(ColumnInfo),
				cbTableCfg := SIZEOF(ColumnInfo))
	THEN
		xCria := FALSE;
	END_IF

END_IF
END_ACTION

END_FUNCTION_BLOCK

// FBs/Partidas/FB_CriaTabelaEMotoresParaInterlock
{attribute 'hide_all_locals'}
FUNCTION_BLOCK FB_CriaTabelaEMotoresParaInterlock
VAR_IN_OUT
	Motor : ARRAY[*] OF st_Partida;
END_VAR
VAR_INPUT
	xCriaTabela		: BOOL;
	iNumeroDataBase	: INT		:= 1;
	sNomeDataBase	: STRING	:= 'motoresconfig';
END_VAR
VAR_OUTPUT
	xOcupado : BOOL;
END_VAR
VAR
	i				: INT;
	xGeraMoto		: BOOL;
	diParteBaixa	: DINT;
	diParteAlta		: DINT;

	//Grava valores
	xGravando		: BOOL;
	rtEscrita		: R_TRIG;
	xEscreve		: BOOL;
	EstruturaBanco	: ST_ConfigMotorDB;
	xEscreveAux		: BOOL;
	sAux			: ARRAY[1..50] OF STRING(80);
	fbPLCDBWrite	: FB_PLCDBWriteEvt(sNetID := '', tTimeout := T#30S); //Bloco para gravar no banco de dados

	ColumnNamesGrava : ARRAY[0..27] OF STRING(50) := ['Motor',
														'Tag',
														'Funcao',

														'InvIT1A',
														'IT1A',
														'OPIT1',
														'InvIT1B',
														'IT1B',

														'InvIT2A',
														'IT2A',
														'OPIT2',
														'InvIT2B',
														'IT2B',

														'InvIT3A',
														'IT3A',
														'OPIT3',
														'InvIT3B',
														'IT3B',

														'InvIT4A',
														'IT4A',
														'OPIT4',
														'InvIT4B',
														'IT4B',

														'Emerg1',
														'Emerg2',
														'Emerg3',
														'Emerg4',
														'Timestamp'
														];

	//Cria table
	rtCria			: R_TRIG;
	xCria			: BOOL;
	fbPLCDBCreate	: FB_PLCDBCreateEvt(sNetID := '', tTimeout := T#30S);

	ColumnInfo :
		ARRAY[0..27] OF ST_ColumnInfo
		:= [(sName := 'Motor', eType := E_ColumnType.BigInt, nLength := 8, sProperty := 'IDENTITY(1,1)'),
				(sName := 'Tag', eType := E_ColumnType.NVarChar, nLength := 80, sProperty := 'DEFAULT $'SEMTAG$''),
				(sName := 'Funcao', eType := E_ColumnType.NVarChar, nLength := 80, sProperty := 'DEFAULT $'NADA$''),

				(sName := 'InvIT1A', eType := E_ColumnType.SmallInt, nLength := 2, sProperty := 'DEFAULT 0'),	//Inverte o interlock 1A
				(sName := 'IT1A', eType := E_ColumnType.NVarChar, nLength := 80, sProperty := 'DEFAULT $'-$''),	//TAG do Interlock 1A
				(sName := 'OPIT1', eType := E_ColumnType.SmallInt, nLength := 2, sProperty := 'DEFAULT 0'),		//Operação entre o interlock 1 A e B
				(sName := 'InvIT1B', eType := E_ColumnType.SmallInt, nLength := 2, sProperty := 'DEFAULT 0'),	//Inverte o interlock 1B
				(sName := 'IT1B', eType := E_ColumnType.NVarChar, nLength := 80, sProperty := 'DEFAULT $'-$''),	// TAG do Interlock 1B

				(sName := 'InvIT2A', eType := E_ColumnType.SmallInt, nLength := 2, sProperty := 'DEFAULT 0'),	//Inverte o interlock 2A
				(sName := 'IT2A', eType := E_ColumnType.NVarChar, nLength := 80, sProperty := 'DEFAULT $'-$''),	//TAG do Interlock 2A
				(sName := 'OPIT2', eType := E_ColumnType.SmallInt, nLength := 2, sProperty := 'DEFAULT 0'),		//Operação entre o interlock 2 A e B
				(sName := 'InvIT2B', eType := E_ColumnType.SmallInt, nLength := 2, sProperty := 'DEFAULT 0'),	//Inverte o interlock 2B
				(sName := 'IT2B', eType := E_ColumnType.NVarChar, nLength := 80, sProperty := 'DEFAULT $'-$''),	// TAG do Interlock 2B

				(sName := 'InvIT3A', eType := E_ColumnType.SmallInt, nLength := 2, sProperty := 'DEFAULT 0'),	//Inverte o interlock 3A
				(sName := 'IT3A', eType := E_ColumnType.NVarChar, nLength := 80, sProperty := 'DEFAULT $'-$''),	//TAG do Interlock 3A
				(sName := 'OPIT3', eType := E_ColumnType.SmallInt, nLength := 2, sProperty := 'DEFAULT 0'),		//Operação entre o interlock 3 A e B
				(sName := 'InvIT3B', eType := E_ColumnType.SmallInt, nLength := 2, sProperty := 'DEFAULT 0'),	//Inverte o interlock 3B
				(sName := 'IT3B', eType := E_ColumnType.NVarChar, nLength := 80, sProperty := 'DEFAULT $'-$''),	// TAG do Interlock 3B

				(sName := 'InvIT4A', eType := E_ColumnType.SmallInt, nLength := 2, sProperty := 'DEFAULT 0'),	//Inverte o interlock 4A
				(sName := 'IT4A', eType := E_ColumnType.NVarChar, nLength := 80, sProperty := 'DEFAULT $'-$''),	//TAG do Interlock 4A
				(sName := 'OPIT4', eType := E_ColumnType.SmallInt, nLength := 2, sProperty := 'DEFAULT 0'),		//Operação entre o interlock 4 A e B
				(sName := 'InvIT4B', eType := E_ColumnType.SmallInt, nLength := 2, sProperty := 'DEFAULT 0'),	//Inverte o interlock 4B
				(sName := 'IT4B', eType := E_ColumnType.NVarChar, nLength := 80, sProperty := 'DEFAULT $'-$''),	// TAG do Interlock 4B

				(sName := 'Emerg1', eType := E_ColumnType.NVarChar, nLength := 80, sProperty := 'DEFAULT $'-$''),		//Emergencia 1
				(sName := 'Emerg2', eType := E_ColumnType.NVarChar, nLength := 80, sProperty := 'DEFAULT $'-$''),		//Emergencia 2
				(sName := 'Emerg3', eType := E_ColumnType.NVarChar, nLength := 80, sProperty := 'DEFAULT $'-$''),		//Emergencia 3
				(sName := 'Emerg4', eType := E_ColumnType.NVarChar, nLength := 80, sProperty := 'DEFAULT $'-$''),		//Emergencia 4
			
				
				(
				sName := 'Timestamp',
					eType := E_ColumnType.DateTime,
					nLength := 4,
					sProperty := 'DEFAULT CURRENT_TIMESTAMP ON UPDATE CURRENT_TIMESTAMP')];
END_VAR



IF xLicensaValida651641iih THEN
	
	GeraTabela();
	GeraOsMotores();

END_IF

ACTION GeraOsMotores:

diParteBaixa	:= LOWER_BOUND(Motor, 1);
diParteAlta		:= UPPER_BOUND(Motor, 1);

IF xGeraMoto THEN

	xEscreve := TRUE;
	rtEscrita(CLK := xEscreve, Q =>);

	IF rtEscrita.q THEN
		xEscreveAux						:= TRUE;
		EstruturaBanco.Motor			:= DINT_TO_LINT(diParteBaixa + i);
		EstruturaBanco.Tag				:= CONCAT('MI', TO_STRING(i));
	END_IF

	IF xEscreveAux THEN
		IF fbPLCDBWrite.WriteStruct
			(
				hDBID := INT_TO_UDINT(iNumeroDataBase),
					sTableName := sNomeDataBase,
					pRecord := ADR(EstruturaBanco),
					cbRecord := SIZEOF(EstruturaBanco),
					pColumnNames := ADR(ColumnNamesGrava),
					cbColumnNames := SIZEOF(ColumnNamesGrava))
		THEN
			xEscreve := FALSE;
			rtEscrita(CLK := xEscreve, Q =>);
			xEscreveAux	:= FALSE;
			i			:= i + 1;

			IF i > diParteAlta THEN
				xGeraMoto	:= FALSE;
				xOcupado	:= FALSE;
			END_IF
		ELSE
			IF fbPLCDBWrite.bError THEN
				IF fbPLCDBWrite.ipTcResult.nEventId = 61 THEN
					xCriaTabela := TRUE;
				END_IF
			END_IF
		END_IF
	END_IF

END_IF
END_ACTION

ACTION GeraTabela:

rtCria(CLK := xCriaTabela, Q =>);

IF rtCria.q THEN
	xCria		:= TRUE;
	xOcupado	:= TRUE;
END_IF

IF xCria THEN

	IF fbPLCDBCreate.Table
		(
			hDBID := INT_TO_UDINT(iNumeroDataBase),
				sTableName := sNomeDataBase,
				pTableCfg := ADR(ColumnInfo),
				cbTableCfg := SIZEOF(ColumnInfo))
	THEN
		xCria		:= FALSE;
		xCriaTabela	:= FALSE;
		xGeraMoto	:= TRUE;
		i			:= 1;
	END_IF

END_IF
END_ACTION

END_FUNCTION_BLOCK

// FBs/Sensores/FB_AtualizaTag
{attribute 'hide_all_locals'}
FUNCTION_BLOCK FB_AtualizaTag
VAR_INPUT
	sPayload		: STRING;
	sTag			: STRING;
	iID				: INT;
	xCriaTabela		: BOOL;
	iNumeroDataBase	: INT := 1;
	sNomeDataBase	: STRING;
END_VAR
VAR_OUTPUT
END_VAR
VAR
	//Criar tabela	
	rtCria			: R_TRIG;
	xCria			: BOOL;
	fbPLCDBCreate	: FB_PLCDBCreateEvt(sNetID := '', tTimeout := T#30S);
	ColumnInfo 		: ARRAY[0..3] OF ST_ColumnInfo := [(sName := 'ID', eType := E_ColumnType.BigInt, nLength := 8, sProperty := 'IDENTITY(1,1)'),
													(sName := 'Tag', eType := E_ColumnType.NVarChar, nLength := 80, sProperty := 'DEFAULT $'SEMTAG$''),
													(sName := 'Payload', eType := E_ColumnType.NVarChar, nLength := 80, sProperty := 'DEFAULT $'NADA$''),
													(sName := 'Timestamp', eType := E_ColumnType.DateTime, nLength := 4, sProperty := 'DEFAULT CURRENT_TIMESTAMP ON UPDATE CURRENT_TIMESTAMP')];
												
	//Atualiza									
	xAtualiza : BOOL;	
									
												
	iEstado : INT := 1;
	i : INT;

	sStatusAnterior	: STRING := sPayload;	
	
	arrConcat	: ARRAY[1..15] OF STRING(255);
	arrConcat2	: ARRAY[1..15] OF STRING(255);

	
	fbPLCDBCmd			: FB_PLCDBCmdEvt(sNetID := '', tTimeout := T#30S);
	fbSqlCommand		: FB_SQLCommandEvt(sNetID := '', tTimeout := T#30S);
	fbSQLDatabase		: FB_SQLDatabaseEvt(sNetID := '', tTimeout := T#30S);
	sCmd				: STRING(1000);
	sCmd1				: STRING(255);
	sCmd2				: STRING(255);
	sCmdUpdate			: STRING(1000);
	sMensagemErro1 		: STRING;
	xAberto : BOOL;
	
	FirstScan	: BOOL	:= TRUE;
END_VAR

IF sPayload <> sStatusAnterior THEN
	sStatusAnterior := sPayload;
	xAtualiza := TRUE;
END_IF


IF FirstScan THEN
	xAtualiza := FALSE;
END_IF

GeraTabela();
Atualiza();

FirstScan := FALSE;

ACTION Atualiza:

CASE iEstado OF
	1: //Esperando
		IF xAtualiza THEN
			IF xAberto THEN
				iEstado := 3;
			ELSE
				iEstado := 2;
			END_IF
		END_IF

	2: //abre conexao
		IF fbSqlDatabase.Connect(int_to_udint(iNumeroDataBase)) THEN
			IF fbSqlDatabase.bError THEN
				IF fbSqlDatabase.ipTcResult.nEventId = 1828 THEN
					// se der isso ele nao fica tentando e gerando uma caralhada de erro pq nao tem a lisença
					iEstado := 0;
				ELSE
					iEstado := 2;
				END_IF
			ELSE
				IF fbSqlDatabase.bConnected THEN
					iEstado := 3;
					xAberto := TRUE;
				ELSE
					iEstado := 5;
					xAberto := FALSE;
				END_IF
			END_IF
		END_IF
	
	3:
		IF fbSqlDatabase.CreateCmd(ADR(fbSqlCommand)) THEN
			IF fbSqlDatabase.bError THEN
				iEstado := 3;
			ELSE
				iEstado := 4;
			END_IF
		END_IF
	

	4: // le o role
	
	//UPDATE `maximo`.`sistema` SET `Status` = 'Desligado' WHERE (`ID` = '1');
		
		arrConcat[1] := 'INSERT INTO geral.';
		arrConcat[2] := sNomeDataBase;
		arrConcat[3] := ' (ID,Tag,Payload) VALUES("';
		arrConcat[4] := TO_STRING(iID);
		arrConcat[5] := '","';
		arrConcat[6] := sTag;
		arrConcat[7] := '","';
		arrConcat2[1] := sPayload;
		arrConcat2[2] := '") ON DUPLICATE KEY UPDATE Tag="';
		arrConcat2[3] := sTag;
		arrConcat2[4] := '", Payload="';
		arrConcat2[5] := sPayload;
		arrConcat2[6] := '";';
	
		
		sCmd1 := F_ConcatArray(sArray:= arrConcat);
		sCmd2 := F_ConcatArray(sArray:= arrConcat2);
		
		CONCAT2(pSrcString1:= ADR(sCmd1), pSrcString2:= ADR(sCmd2), pDstString:= ADR(sCmd), nDstSize:= 10000);
		// call functionblock
		IF xAtualiza THEN		
			IF fbSQLCommand.Execute(pSQLCmd := ADR(sCmd), cbSQLCmd := SIZEOF(sCmd))
			THEN
				IF fbSQLCommand.bError THEN
					IF fbSQLCommand.ipTcResult.nEventId = 61 THEN
					// se der isso ele nao fica tentando e gerando uma caralhada de erro pq nao tem a lisença
					iEstado := 1;
						xCriaTabela := TRUE;
					ELSE
						iEstado := 2;
					END_IF
					sMensagemErro1 := 'Nao conseguiu a tag';
				ELSE
					sMensagemErro1	:= 'Conseguiu a tag';
				END_IF
				iEstado := 5;
				xAtualiza := FALSE;
			END_IF
		END_IF

	5: // FechaConexao conexao
		IF fbSqlDatabase.Disconnect() THEN

			xAtualiza := FALSE;

			IF fbSqlDatabase.bError THEN
				iEstado := 1;
			ELSE
				iEstado := 1;
				xAberto := FALSE;
			END_IF
		END_IF
END_CASE
END_ACTION

ACTION GeraTabela:

rtCria(CLK := xCriaTabela, Q =>);

IF rtCria.q THEN
	xCria := TRUE;
END_IF

IF xCria THEN

	IF fbPLCDBCreate.Table(
			hDBID := INT_TO_UDINT(iNumeroDataBase),
			sTableName := sNomeDataBase,
			pTableCfg := ADR(ColumnInfo),
			cbTableCfg := SIZEOF(ColumnInfo))
	THEN
		xCria := FALSE;
		xCriaTabela := FALSE;
	END_IF

END_IF
END_ACTION

END_FUNCTION_BLOCK

// FBs/Sensores/FB_CriaTabelaSensores
{attribute 'hide_all_locals'}
FUNCTION_BLOCK FB_CriaTabelaSensores
VAR_IN_OUT
	Sensores : ARRAY[*] OF st_SensorDigital;
END_VAR
VAR_INPUT
	xCriaTabela		: BOOL;
	iNumeroDataBase	: INT		:= 1;
	sNomeDataBase	: STRING	:= 'SensoresConfig';
	sInicoNome : STRING := 'SO';
END_VAR
VAR_OUTPUT
	xOcupado : BOOL;
END_VAR
VAR
	i				: INT;
	xGeraMoto		: BOOL;
	diParteBaixa	: DINT;
	diParteAlta		: DINT;

	//Grava valores
	xGravando		: BOOL;
	rtEscrita		: R_TRIG;
	xEscreve		: BOOL;
	EstruturaBanco	: st_LeConfigSensorNoBanco;
	xEscreveAux		: BOOL;
	sAux			: ARRAY[1..50] OF STRING(80);
	fbPLCDBWrite	: FB_PLCDBWriteEvt(sNetID := '', tTimeout := T#30S); //Bloco para gravar no banco de dados

	ColumnNamesGrava : ARRAY[0..2] OF STRING(50) := ['Sensor',
													'Tag',
													'Funcao'];

	//Cria table
	rtCria			: R_TRIG;
	xCria			: BOOL;
	fbPLCDBCreate	: FB_PLCDBCreateEvt(sNetID := '', tTimeout := T#30S);

	ColumnInfo :
		ARRAY[0..3] OF ST_ColumnInfo
		:= [(sName := 'Sensor', eType := E_ColumnType.BigInt, nLength := 8, sProperty := 'IDENTITY(1,1)'),
				(sName := 'Tag', eType := E_ColumnType.NVarChar, nLength := 80, sProperty := 'DEFAULT $'SEMTAG$''),
				(sName := 'Funcao', eType := E_ColumnType.NVarChar, nLength := 80, sProperty := 'DEFAULT $'NADA$''),
				(
				sName := 'Timestamp',
					eType := E_ColumnType.DateTime,
					nLength := 4,
					sProperty := 'DEFAULT CURRENT_TIMESTAMP ON UPDATE CURRENT_TIMESTAMP')];
END_VAR

IF xLicensaValida651641iih THEN
	
	GeraTabela();
	GeraOsSensores();
END_IF

ACTION GeraOsSensores:

diParteBaixa	:= LOWER_BOUND(Sensores, 1);
diParteAlta		:= UPPER_BOUND(Sensores, 1);

IF xGeraMoto THEN

	xEscreve := TRUE;
	rtEscrita(CLK := xEscreve, Q =>);

	IF rtEscrita.q THEN
		xEscreveAux						:= TRUE;
		EstruturaBanco.Sensor.dwLowPart	:= DINT_TO_DWORD(diParteBaixa + i);
		EstruturaBanco.Tag				:= CONCAT(sInicoNome, TO_STRING(i));
	END_IF

	IF xEscreveAux THEN
		IF fbPLCDBWrite.WriteStruct
			(
				hDBID := INT_TO_UDINT(iNumeroDataBase),
					sTableName := sNomeDataBase,
					pRecord := ADR(EstruturaBanco),
					cbRecord := SIZEOF(EstruturaBanco),
					pColumnNames := ADR(ColumnNamesGrava),
					cbColumnNames := SIZEOF(ColumnNamesGrava))
		THEN
			xEscreve := FALSE;
			rtEscrita(CLK := xEscreve, Q =>);
			xEscreveAux	:= FALSE;
			i			:= i + 1;

			IF i > diParteAlta THEN
				xGeraMoto	:= FALSE;
				xOcupado	:= FALSE;
			END_IF
		END_IF
	END_IF

END_IF
END_ACTION

ACTION GeraTabela:

rtCria(CLK := xCriaTabela, Q =>);

IF rtCria.q THEN
	xCria		:= TRUE;
	xOcupado	:= TRUE;
END_IF

IF xCria THEN

	IF fbPLCDBCreate.Table
		(
			hDBID := INT_TO_UDINT(iNumeroDataBase),
				sTableName := sNomeDataBase,
				pTableCfg := ADR(ColumnInfo),
				cbTableCfg := SIZEOF(ColumnInfo))
	THEN
		IF NOT fbPLCDBCreate.bError THEN
			xCria		:= FALSE;
			xCriaTabela	:= FALSE;
			xGeraMoto	:= TRUE;
			i			:= 1;
		ELSE
			xCria		:= FALSE;
			xCriaTabela	:= FALSE;
		END_IF
	END_IF

END_IF
END_ACTION

END_FUNCTION_BLOCK

// FBs/Sensores/FB_DBComparaSensor
{attribute 'hide_all_locals'}
FUNCTION_BLOCK FB_DBComparaSensor
VAR_INPUT
	Sensores 		: st_ComparaAnalogico;	// st do sensor analogico lido e manual
	sNomeDataBase	: STRING;				// nome do sensor para a criação da tabela
	iNumeroDataBase	: INT		:= 1;		// id do database	
	xCriaTabela		: BOOL;					// tenta criar a tabela
	tTempoDeAmostra	: TIME;					// tempo entre cada amostra
END_VAR
VAR_OUTPUT
	xOcupado : BOOL;
END_VAR
VAR
	//Cria table
	rtCria			: R_TRIG;
	xCria			: BOOL;
	fbPLCDBCreate	: FB_PLCDBCreateEvt(sNetID := '', tTimeout := T#30S);
	
	ColumnInfo : ARRAY[0..4] OF ST_ColumnInfo := [(sName := 'ID', eType := E_ColumnType.BigInt, nLength := 8, sProperty := 'IDENTITY(1,1)'),
												(sName := 'rAnalogicoLido', eType := E_ColumnType.REAL_, nLength := 4),
												(sName := 'rAnalogicoManual', eType := E_ColumnType.REAL_, nLength := 4),
												(sName := 'rDiferenca', eType := E_ColumnType.REAL_, nLength := 4),
												(
				sName := 'Timestamp',
					eType := E_ColumnType.DateTime,
					nLength := 4,
					sProperty := 'DEFAULT CURRENT_TIMESTAMP ON UPDATE CURRENT_TIMESTAMP')];

	ColumnNamesGrava : ARRAY[0..3] OF STRING(50) := ['ID',
												'rAnalogicoLido',
												'rAnalogicoManual',
												'rDiferenca'];
	
	//Grava valores
	xEscreve			: BOOL;
	fbPLCDBWrite		: FB_PLCDBWriteEvt(sNetID := '', tTimeout := T#30S); //Bloco para gravar no banco de dados
	fbPLCDBCmd			: FB_PLCDBCmdEvt(sNetID := '', tTimeout := T#30S);
	fbSqlCommand		: FB_SQLCommandEvt(sNetID := '', tTimeout := T#30S);
	fbSQLDatabase		: FB_SQLDatabaseEvt(sNetID := '', tTimeout := T#30S);
	sCmd				: STRING(1000);
	sCmdUpdate			: STRING(1000);
	sMensagemErro1 		: STRING;
	xAberto 			: BOOL;
	rtComecaEscrever 	: R_TRIG;
	iEstado 			:	INT := 1;
	tonEscrita			: TON;
	rtSalva				: R_TRIG;
	rAnalogicoManual	: REAL;
	rDiferenca			: REAL;
	xSalva				: BOOL;
END_VAR

IF xLicensaValida651641iih THEN
		
	
	/// Criado por Augusto Cazanelli em 11/05/2022
	
	tonEscrita.IN := TRUE;
	
	rtSalva(CLK:= Sensores.xSalva, Q=> );
	
	IF tonEscrita.q OR rtSalva.Q THEN
		IF (rtSalva.Q) THEN
			rAnalogicoManual := Sensores.rAnalogicoManual;
			xSalva := TRUE;
		ELSE
			rAnalogicoManual := 0;
		END_IF
		
		rDiferenca := Sensores.rAnalogicoLido - rAnalogicoManual; 	
		tonEscrita.IN	:= FALSE;
		xEscreve		:= TRUE;
	END_IF
	
	tonEscrita(PT := tTempoDeAmostra, Q =>, ET =>);
	
	GeraTabela();
	GravaValores();

END_IF

ACTION GeraTabela:

rtCria(CLK := xCriaTabela, Q =>);

IF rtCria.q THEN
	xCria		:= TRUE;
	xOcupado	:= TRUE;
END_IF

IF xCria THEN

	IF fbPLCDBCreate.Table
		(
			hDBID := INT_TO_UDINT(iNumeroDataBase),
				sTableName := sNomeDataBase,
				pTableCfg := ADR(ColumnInfo),
				cbTableCfg := SIZEOF(ColumnInfo))
	THEN
		IF NOT fbPLCDBCreate.bError THEN
			xCria		:= FALSE;
			xCriaTabela	:= FALSE;
		ELSE
			xCria		:= FALSE;
			xCriaTabela	:= FALSE;
		END_IF
	END_IF

END_IF
END_ACTION

ACTION GravaValores:

CASE iEstado OF
	1: //Esperando
		IF xEscreve THEN
			IF xAberto THEN
				iEstado := 3;	//Caso para abrir a conexão
			ELSE
				iEstado := 2;	//Caso em que a conexão já foi aberta
			END_IF
		END_IF

	2: //abre conexao
		IF fbSqlDatabase.Connect(int_to_udint(iNumeroDataBase)) THEN
			IF fbSqlDatabase.bError THEN
				IF fbSqlDatabase.ipTcResult.nEventId = 1828 THEN
					// se der isso ele nao fica tentando e gerando uma caralhada de erro pq nao tem a lisença
					iEstado := 0;
				ELSE
					iEstado := 2;
				END_IF
			ELSE
				IF fbSqlDatabase.bConnected THEN
					iEstado := 3;
					xAberto := TRUE;
				ELSE
					iEstado := 5;
					xAberto := FALSE;
				END_IF
			END_IF
		END_IF
	
	3:
		IF fbSqlDatabase.CreateCmd(ADR(fbSqlCommand)) THEN
			IF fbSqlDatabase.bError THEN
				iEstado := 3;
			ELSE
				iEstado := 4;
			END_IF
		END_IF
	

	4: // le o role
	
		// call functionblock
		IF xEscreve THEN	
		
		IF xSalva THEN
				//'INSERT INTO geral.S01 (rAnalogicoLido, rAnalogicoManual, rDiferenca) VALUES (Sensores.rAnalogicoLido, Sensores.rAnalogicoManual, Sensores.rDiferenca);'	
			sCmd := CONCAT(
					CONCAT(
					CONCAT(
					CONCAT(
					CONCAT(
					CONCAT(
					CONCAT(
					CONCAT(
					'INSERT INTO geral.', sNomeDataBase),
					'(rAnalogicoLido, rAnalogicoManual, rDiferenca) VALUES ('),
					TO_STRING(Sensores.rAnalogicoLido)),
					' , '),
					TO_STRING(rAnalogicoManual)),
					' , '),
					TO_STRING(rDiferenca)),
					');');	
					
					xSalva := FALSE;
		ELSE
							//'INSERT INTO geral.S01 (rAnalogicoLido, rAnalogicoManual, rDiferenca) VALUES (Sensores.rAnalogicoLido, Sensores.rAnalogicoManual, Sensores.rDiferenca);'	
			sCmd := CONCAT(
					CONCAT(
					CONCAT(
					CONCAT(
					CONCAT(
					CONCAT(
					'INSERT INTO geral.', sNomeDataBase),
					'(rAnalogicoLido, rDiferenca) VALUES ('),
					TO_STRING(Sensores.rAnalogicoLido)),
					' , '),
					TO_STRING(rDiferenca)),
					');');	
		END_IF
		
				
			IF fbSQLCommand.Execute(pSQLCmd := ADR(sCmd), cbSQLCmd := SIZEOF(sCmd))
			THEN
				IF fbSQLCommand.bError THEN
					IF fbSQLCommand.ipTcResult.nEventId = 61 THEN
					// Esse erro acontece quando o database não tá criado, nesse caso ele tenta criar
					iEstado := 1;
						xCriaTabela := TRUE;
					ELSE
						iEstado := 2;
					END_IF
					sMensagemErro1 := 'Nao conseguiu a tag';
				ELSE
					sMensagemErro1	:= 'Conseguiu a tag';
				END_IF
				iEstado := 5;
				xEscreve := FALSE;
			END_IF
		END_IF

	5: // FechaConexao conexao
		IF fbSqlDatabase.Disconnect() THEN

			xEscreve := FALSE;

			IF fbSqlDatabase.bError THEN
				iEstado := 1;
			ELSE
				iEstado := 1;
				xAberto := FALSE;
			END_IF
		END_IF
END_CASE
END_ACTION

END_FUNCTION_BLOCK

// FBs/Sensores/FB_HistoricoSQL
{attribute 'hide_all_locals'}
FUNCTION_BLOCK FB_HistoricoSQL
VAR_INPUT
	rValor			: REAL;
	tTempoDeAmostra	: TIME;
	xCriaTabela		: BOOL;
	iNumeroDataBase	: INT := 1;
	sNomeDataBase	: STRING	:= 'LeitorAnalogico1';
END_VAR
VAR_OUTPUT
END_VAR
VAR
	iEstado : INT := 1;
	rtCria			: R_TRIG;
	xCria			: BOOL;
	fbPLCDBCreate	: FB_PLCDBCreateEvt(sNetID := '', tTimeout := T#30S);

	ColumnInfo : ARRAY[0..2] OF ST_ColumnInfo := [(sName := 'ID', eType := E_ColumnType.BigInt, nLength := 8, sProperty := 'IDENTITY(1,1)'),
												(sName := 'Valor', eType := E_ColumnType.Float, nLength := 8),
												(
				sName := 'Timestamp',
					eType := E_ColumnType.DateTime,
					nLength := 4,
					sProperty := 'DEFAULT CURRENT_TIMESTAMP ON UPDATE CURRENT_TIMESTAMP')];


	tonEscrita	: TON;
	xEscreve	: BOOL;


	xAtualiza : BOOL;
	ColumnNamesLe : ARRAY[0..2] OF STRING(50) := ['ID',
												'Valor',
												'Timestamp'];
	iTamanhoHistorico : DINT;

	i : INT;
	
	fbPLCDBCmd			: FB_PLCDBCmdEvt(sNetID := '', tTimeout := T#30S);
	fbSqlCommand		: FB_SQLCommandEvt(sNetID := '', tTimeout := T#30S);
	fbSQLDatabase		: FB_SQLDatabaseEvt(sNetID := '', tTimeout := T#30S);
	sCmd				: STRING(1000);
	sCmdUpdate			: STRING(1000);
	sMensagemErro1 		: STRING;
	xAberto : BOOL;
	rtComecaEscrever : R_TRIG;
END_VAR

IF xLicensaValida651641iih THEN
	

	tonEscrita.IN := TRUE;
	
	IF tonEscrita.q THEN
	tonEscrita.IN	:= FALSE;
	xEscreve		:= TRUE;
	END_IF
	
	tonEscrita(PT := tTempoDeAmostra, Q =>, ET =>);
	
	GeraTabela();
	GravaHistorico();

END_IF

ACTION GeraTabela:

rtCria(CLK := xCriaTabela, Q =>);

IF rtCria.q THEN
	xCria := TRUE;
END_IF

IF xCria THEN

	IF fbPLCDBCreate.Table(
			hDBID := INT_TO_UDINT(iNumeroDataBase),
			sTableName := sNomeDataBase,
			pTableCfg := ADR(ColumnInfo),
			cbTableCfg := SIZEOF(ColumnInfo))
	THEN
		xCria := FALSE;
		xCriaTabela := FALSE;
	END_IF

END_IF
END_ACTION

ACTION GravaHistorico:

CASE iEstado OF
	1: //Esperando
		IF xEscreve THEN
			IF xAberto THEN
				iEstado := 3;
			ELSE
				iEstado := 2;
			END_IF
		END_IF

	2: //abre conexao
		IF fbSqlDatabase.Connect(int_to_udint(iNumeroDataBase)) THEN
			IF fbSqlDatabase.bError THEN
				IF fbSqlDatabase.ipTcResult.nEventId = 1828 THEN
					// se der isso ele nao fica tentando e gerando uma caralhada de erro pq nao tem a lisença
					iEstado := 0;
				ELSE
					iEstado := 2;
				END_IF
			ELSE
				IF fbSqlDatabase.bConnected THEN
					iEstado := 3;
					xAberto := TRUE;
				ELSE
					iEstado := 5;
					xAberto := FALSE;
				END_IF
			END_IF
		END_IF
	
	3:
		IF fbSqlDatabase.CreateCmd(ADR(fbSqlCommand)) THEN
			IF fbSqlDatabase.bError THEN
				iEstado := 3;
			ELSE
				iEstado := 4;
			END_IF
		END_IF
	

	4: // le o role

		sCmd := CONCAT(CONCAT(CONCAT(CONCAT('INSERT INTO geral.', sNomeDataBase),'(Valor) Value ('),TO_STRING(rValor)), ');');	


		// call functionblock
		IF xEscreve THEN		
			IF fbSQLCommand.Execute(pSQLCmd := ADR(sCmd), cbSQLCmd := SIZEOF(sCmd))
			THEN
				IF fbSQLCommand.bError THEN
					IF fbSQLCommand.ipTcResult.nEventId = 61 THEN
					// se der isso ele nao fica tentando e gerando uma caralhada de erro pq nao tem a lisença
					iEstado := 1;
						xCriaTabela := TRUE;
					ELSE
						iEstado := 2;
					END_IF
					sMensagemErro1 := 'Nao conseguiu a tag';
				ELSE
					sMensagemErro1	:= 'Conseguiu a tag';
				END_IF
				iEstado := 5;
				xEscreve := FALSE;
			END_IF
		END_IF

	5: // FechaConexao conexao
		IF fbSqlDatabase.Disconnect() THEN

			xEscreve := FALSE;

			IF fbSqlDatabase.bError THEN
				iEstado := 1;
			ELSE
				iEstado := 1;
				xAberto := FALSE;
			END_IF
		END_IF
END_CASE
END_ACTION

END_FUNCTION_BLOCK

// FBs/Sensores/FB_HistoricoTag
{attribute 'hide_all_locals'}
FUNCTION_BLOCK FB_HistoricoTag
VAR_INPUT
	rValor			: REAL;
	sTag			: STRING;
	tTempoDeAmostra	: TIME;
	xCriaTabela		: BOOL;
	iNumeroDataBase	: INT := 1;
	sNomeDataBase	: STRING;
END_VAR
VAR_OUTPUT
END_VAR
VAR
	//Criar tabela	
	rtCria			: R_TRIG;
	xCria			: BOOL;
	fbPLCDBCreate	: FB_PLCDBCreateEvt(sNetID := '', tTimeout := T#30S);
	ColumnInfo 		: ARRAY[0..2] OF ST_ColumnInfo := [(sName := 'Tag', eType := E_ColumnType.NVarChar, nLength := 80, sProperty := 'DEFAULT $'SEMTAG$''),
													(sName := 'Payload', eType := E_ColumnType.REAL_, nLength := 4),
													(sName := 'Timestamp', eType := E_ColumnType.DateTime, nLength := 4, sProperty := 'DEFAULT CURRENT_TIMESTAMP ON UPDATE CURRENT_TIMESTAMP')];
												
	//Atualiza									
	xAtualiza : BOOL;																		
	iEstado : INT := 1;
	i : INT;
	arrConcat	: ARRAY[1..15] OF STRING(255);
	arrConcat2	: ARRAY[1..15] OF STRING(255);	
	fbPLCDBCmd			: FB_PLCDBCmdEvt(sNetID := '', tTimeout := T#30S);
	fbSqlCommand		: FB_SQLCommandEvt(sNetID := '', tTimeout := T#30S);
	fbSQLDatabase		: FB_SQLDatabaseEvt(sNetID := '', tTimeout := T#30S);
	sCmd				: STRING(1000);
	sCmd1				: STRING(255);
	sCmd2				: STRING(255);
	sCmdUpdate			: STRING(1000);
	sMensagemErro1 		: STRING;
	xAberto 			: BOOL;
	tonEscrita			: Tc2_Standard.TON;
	FirstScan	: BOOL	:= TRUE;
END_VAR


//xAtualiza := TRUE;
tonEscrita.IN := TRUE;

IF tonEscrita.q THEN
	tonEscrita.IN	:= FALSE;
	xAtualiza		:= TRUE;
END_IF

tonEscrita(PT := tTempoDeAmostra, Q =>, ET =>);


IF FirstScan THEN
	xAtualiza := FALSE;
END_IF

GeraTabela();
Atualiza();

FirstScan := FALSE;

ACTION Atualiza:

CASE iEstado OF
	1: //Esperando
		IF xAtualiza THEN
			IF xAberto THEN
				iEstado := 3;
			ELSE
				iEstado := 2;
			END_IF
		END_IF

	2: //abre conexao
		IF fbSqlDatabase.Connect(int_to_udint(iNumeroDataBase)) THEN
			IF fbSqlDatabase.bError THEN
				IF fbSqlDatabase.ipTcResult.nEventId = 1828 THEN
					// se der isso ele nao fica tentando e gerando uma caralhada de erro pq nao tem a lisença
					iEstado := 0;
				ELSE
					iEstado := 2;
				END_IF
			ELSE
				IF fbSqlDatabase.bConnected THEN
					iEstado := 3;
					xAberto := TRUE;
				ELSE
					iEstado := 5;
					xAberto := FALSE;
				END_IF
			END_IF
		END_IF
	
	3:
		IF fbSqlDatabase.CreateCmd(ADR(fbSqlCommand)) THEN
			IF fbSqlDatabase.bError THEN
				iEstado := 3;
			ELSE
				iEstado := 4;
			END_IF
		END_IF
	

	4: // le o role
	
	//UPDATE `maximo`.`sistema` SET `Status` = 'Desligado' WHERE (`ID` = '1');
		
		arrConcat[1] := 'INSERT INTO geral.';
		arrConcat[2] := sNomeDataBase;
		arrConcat[3] := ' (Tag,Payload) VALUES("';
		arrConcat[4] := sTag;
		arrConcat[5] := '",';
		arrConcat2[1] := TO_STRING(rValor);
		arrConcat2[2] := ');';

	
		
		sCmd1 := F_ConcatArray(sArray:= arrConcat);
		sCmd2 := F_ConcatArray(sArray:= arrConcat2);
		
		CONCAT2(pSrcString1:= ADR(sCmd1), pSrcString2:= ADR(sCmd2), pDstString:= ADR(sCmd), nDstSize:= 10000);
		// call functionblock
		IF xAtualiza THEN		
			IF fbSQLCommand.Execute(pSQLCmd := ADR(sCmd), cbSQLCmd := SIZEOF(sCmd))
			THEN
				IF fbSQLCommand.bError THEN
					IF fbSQLCommand.ipTcResult.nEventId = 61 THEN
					// se der isso ele nao fica tentando e gerando uma caralhada de erro pq nao tem a lisença
					iEstado := 1;
						xCriaTabela := TRUE;
					ELSE
						iEstado := 2;
					END_IF
					sMensagemErro1 := 'Nao conseguiu a tag';
				ELSE
					sMensagemErro1	:= 'Conseguiu a tag';
				END_IF
				iEstado := 5;
				xAtualiza := FALSE;
			END_IF
		END_IF

	5: // FechaConexao conexao
		IF fbSqlDatabase.Disconnect() THEN

			xAtualiza := FALSE;

			IF fbSqlDatabase.bError THEN
				iEstado := 1;
			ELSE
				iEstado := 1;
				xAberto := FALSE;
			END_IF
		END_IF
END_CASE
END_ACTION

ACTION GeraTabela:

rtCria(CLK := xCriaTabela, Q =>);

IF rtCria.q THEN
	xCria := TRUE;
END_IF

IF xCria THEN

	IF fbPLCDBCreate.Table(
			hDBID := INT_TO_UDINT(iNumeroDataBase),
			sTableName := sNomeDataBase,
			pTableCfg := ADR(ColumnInfo),
			cbTableCfg := SIZEOF(ColumnInfo))
	THEN
		xCria := FALSE;
		xCriaTabela := FALSE;
	END_IF

END_IF
END_ACTION

END_FUNCTION_BLOCK

// FBs/Sensores/FB_IniciaOsBlocosDeSensor
{attribute 'hide_all_locals'}
FUNCTION_BLOCK FB_IniciaOsBlocosDeSensor
VAR_IN_OUT
	sSensor : ARRAY[*] OF st_SensorDigital;
END_VAR
VAR_INPUT
	xInicia : BOOL;
	iNumeroDataBase	: INT		:= 1;
	sNomeDataBase	: STRING	:= 'SensoresConfig';
END_VAR
VAR_OUTPUT
END_VAR
VAR
	fbPLCDBCmd			: FB_PLCDBCmdEvt(sNetID := '', tTimeout := T#60S);
	fbSQLDatabase		: FB_SQLDatabaseEvt(sNetID := '', tTimeout := T#60S);
	sCmd				: STRING(1000);
	sCmdUpdate			: STRING(1000);
	stPara				: ST_ExpParameter;
	TagAProcurar		: STRING(80);
	nRecords			: UDINT;
	xProcuraNaTabela	: BOOL;
	EstruturaBanco		: ARRAY[0..999] OF Teknike_Sensores.st_LeConfigSensorNoBanco;
	xJogaNoInterlock	: BOOL;
	sTag1				: STRING;
	sTag2				: STRING;
	xEMotor				: BOOL;
	sMensagemErro1		: STRING;
	diCimaSensor		: DINT;
	diBaixoSensor		: DINT;

	iEstado	: INT := 1;
	i		: INT;

	iAux : INT;

END_VAR


IF xLicensaValida651641iih THEN
	
	CASE iEstado OF
		1: //Esperando
			IF xInicia THEN
				iEstado := 2;
			END_IF
	
		2: //abre conexao
			IF fbSqlDatabase.Connect(int_to_udint(iNumeroDataBase)) THEN
				IF fbSqlDatabase.bError THEN
					IF fbSqlDatabase.ipTcResult.ipSourceInfo.sName = 'ADSERR_DEVICE_LICENSENOTFOUND' THEN
						// se der isso ele nao fica tentando e gerando uma caralhada de erro pq nao tem a lisença
						iEstado := 0;
					ELSE
						iEstado := 2;
					END_IF
				ELSE
					IF fbSqlDatabase.bConnected THEN
						iEstado := 3;
					END_IF
				END_IF
			END_IF
	
		3: // le o role
			TagAProcurar		:= sTag1;
			stPara.eParaType	:= E_ExpParameterType.STRING_;
			stPara.nParaSize	:= SIZEOF(TagAProcurar);
			stPara.sParaName	:= 'Tag';
	
			diBaixoSensor	:= LOWER_BOUND(sSensor, 1);
			diCimaSensor	:= UPPER_BOUND(sSensor, 1);
	
			// set command with placeholder
			sCmd := CONCAT(CONCAT('SELECT * FROM ',sNomeDataBase),';');
	
			// call functionblock
			IF fbPLCDBCmd.ExecuteDataReturn
				(
					hDBID := 1,
						pExpression := ADR(sCmd),
						cbExpression := SIZEOF(sCmd),
						pData := ADR(TagAProcurar),
						cbData := SIZEOF(TagAProcurar),
						pParameter := ADR(stPara),
						cbParameter := SIZEOF(stPara),
						nStartIndex := 0,
						nRecordCount := DINT_TO_UDINT(diCimaSensor),
						pReturnData := ADR(EstruturaBanco),
						cbReturnData := SIZEOF(EstruturaBanco),
						pRecords := ADR(nRecords))
			THEN
				IF fbPLCDBCmd.bError THEN
					sMensagemErro1 := 'Nao conseguiu a tag';
				ELSE
					sMensagemErro1	:= 'Conseguiu a tag';
					iEstado			:= 4;
	
					FOR i := TO_INT(diBaixoSensor) TO TO_INT(diCimaSensor)-1 DO
						sSensor[i+1].Banco := EstruturaBanco[i];
						sSensor[i].config.sNome_Funcao := CONCAT(CONCAT(sSensor[i].Banco.Tag,' - '),sSensor[i].Banco.Funcao);
					END_FOR
				END_IF
			END_IF
	
		4: // FechaConexao conexao
			IF fbSqlDatabase.Disconnect() THEN
	
				xInicia := FALSE;
	
				IF fbSqlDatabase.bError THEN
					iEstado := 1;
				ELSE
					iEstado := 1;
				END_IF
			END_IF
	END_CASE

END_IF

END_FUNCTION_BLOCK

// POUs/MAIN
PROGRAM MAIN
VAR
	fb1 : FB_ConfigPartidaNoBanco;
	fb2 : FB_CriaTabelaEMotoresParaInterlock;
	fb3 : FB_IniciaOsBlocosDeConfigDoMotor;
	fb4 : FB_CriaTabelaSensores;
	fb5 : FB_IniciaOsBlocosDeSensor;
	fb6 : FB_HistoricoSQL;
	fb7 : FB_KPIPartidasSQL;
	fb8	: FB_DBComparaSensor;
	fb9	: FB_HistogramaSKUsMaisLidas;
	fb10	: FB_CriaTabelaEmergencias;
	fb11	: FB_IniciaOsBlocosDaEmergencia;
	fb12	: FB_IniciaGrupos;
	fb13	: FB_ControleGrupo;
	fb14	: FB_GeraListaInterlocksIHM;
END_VAR

END_PROGRAM

// Project Information/F_GetCompany
// This function has been automatically generated from the project information.
{attribute 'signature_flag' := '1073741824'}
{attribute 'TcGenerated'}
{attribute 'no-analysis'}
FUNCTION F_GetCompany : WSTRING
VAR_INPUT
	
END_VAR

F_GetCompany := "Teknike";

END_FUNCTION

// Project Information/F_GetTitle
// This function has been automatically generated from the project information.
{attribute 'signature_flag' := '1073741824'}
{attribute 'TcGenerated'}
{attribute 'no-analysis'}
FUNCTION F_GetTitle : WSTRING
VAR_INPUT
	
END_VAR

F_GetTitle := "SQL";

END_FUNCTION

// Project Information/F_GetVersion
// This function has been automatically generated from the project information.
{attribute 'signature_flag' := '1073741824'}
{attribute 'TcGenerated'}
{attribute 'no-analysis'}
FUNCTION F_GetVersion : ST_LibVersion
VAR_INPUT
	
END_VAR

F_GetVersion.iMajor := 2;
F_GetVersion.iMinor := 5;
F_GetVersion.iBuild := 8;
F_GetVersion.iRevision := 0;
F_GetVersion.sVersion := '2.5.8';
F_GetVersion.nFlags := 0;

END_FUNCTION
